Fanuc KAREL source: COPY_TPE.kl

PROGRAM T
%NOLOCKGROUP
VAR
 v0 : STRING[40]
 v1 : STRING[40]
 v2 : BOOLEAN
 v3 : INTEGER
BEGIN
 COPY_TPE(v0, v1, v2, v3)
END T
